TYPE STATE:
    STRUCT
        curTime: LREAL;
        dvar_M_a_li AT %Q*: ARRAY[0..4] of DINT;
    END_STRUCT
END_TYPE

(* stored: ProductVersion 3.1.0.18, Version 1.1.0.1 *)
